FUNCTION "FC_Any_ASCII_To_DInt" : VOID
TITLE =%version: 0.06 % CN: 31
//Function:
//Convert a field of ASCII digits to a Double Integer.
//
//Description:
//
//IMPORTANT
//When u use symbolics at the input of type ANY that refer to a variable of the
//type array or structure be aware that the number of array or structure is even
//!
//
//examples: array[1..2]; array[1..4]; array[1..24]; etc.
//
//             t_char   STRUCT
//              |nr_1   BYTE
//              |nr_2   BYTE
//              |nr_3   BYTE
//              |nr_4   BYTE
//
//The any pointer i_ASCII_pnt points to an area which contains an ASCII number.
//When called, this function converts the imported ASCII-number to a double
//integer and returns the result through o_DInteger_number. The ASCII number can
//be of 1 up to 10 bytes. The ASCII number is split into three double integer
//parts. Then the three parts are checked on the physical limit of a double
//integer. This results into an input specification a range of 0..2147483647.
//When the ASCII-number is out of range, the conversion will not be carried out*.
//Contents of the address registers are being remembered during the block call.
//This way the address registers can be used in the current block.
//The output o_RET_VAL contains information about the cause of the errror.
//· Code 0000:
//No error.
//· Code 3115: {information code}
//The area destination of the any pointer is too small (<5 bytes). When the
//integer number is greater than the destination, only the msb's of the integer
//number will be copied.
//. Code 3112: {error code}
//ASCII type is not 3x hex (0 <= x <=  9). BR-bit is set.
//. Code 3111: {error code}
//The double integer number is out of range. BR-bit is set.
//. Code 3113: {error code}
//Data type is neither byte nor char. BR-bit is set.
//. Code 3114: {error code}
//Wrong memory area from any pointer. BR-bit is set.
//
//
//example: '1248365402' (31 32 34 38 33 36 35 34 30 32 hex.)is converted
//into 1248365402
//
//History:
//This version  %created_by:   %
//              %date_created:   %
//              %release: ECS_General_PLC/dev %
//
//Initial version based on the FC_Any_ASCII_To_DInt Rev: 1.11 of the SSS General
//library
//
//Modification History:                                   By:    Date:     Rev:
//----------------------------------------------------  -------  --------  -----
//7324: ECS-P General from the RD to RA for platform    nlHdL    06-07-15   0.06
//15807: Block consistency update IO symbols, comment   nlHdL    18-09-13   0.06
//CR8255 Update internal logging event value            nlcsu    11-11-11   0.05
//CR6415 Remove o_RET_VAL                               nlple    28-09-11   0.04
//CR6341 Update to coding standard                      nlHdL    27-01-11   0.03
//CR6275 Changing compilation number                    nlple    17-01-11   0.02
//Initial revision                                      nlple    14-01-11   0.01
//
FAMILY : General
VERSION : 0.0


VAR_INPUT
  i_ANY_ASCII : ANY ;	//ANY pointer to the ASCII digits
  i_DB_Event_Num : INT ;	//Number of DB event
END_VAR
VAR_OUTPUT
  o_DINT : DINT ;	//Output of the DINT
END_VAR
VAR_TEMP
  t_char : STRUCT 	//Local Copy of the ASCII digits
   nr_1 : BYTE ;
   nr_2 : BYTE ;
   nr_3 : BYTE ;
   nr_4 : BYTE ;
   nr_5 : BYTE ;
   nr_6 : BYTE ;
   nr_7 : BYTE ;
   nr_8 : BYTE ;
   nr_9 : BYTE ;
   nr_10 : BYTE ;
  END_STRUCT ;
  t_DInteger_H : DINT ;	//Double Integer High part: Bytes 1..4
  t_DInteger_M : DINT ;	//Double Integer Medium part: Bytes 5..8
  t_DInteger_L : DINT ;	//Double Integer Low part: Bytes 9..10
  t_ANY_P_ASCII : ANY ;	//Temp of the ANY pointer
  t_DInteger_number : DINT ;	//Temp of Double Integer
  t_ANY_P_Byte_Address : INT ;	//Byte Address of ANY
  t_Data_Type : DWORD ;	//Data Type of ANY
  t_ANY_P_Length : INT ;	//Lenght of ANY
  t_AR1_Store : DWORD ;	//Store for AR1
  t_AR2_Store : DWORD ;	//Store for AR2
  t_Loop_cntr : INT ;	//Loop Counter
  t_Data_Type_Byte : BYTE ;	//Date Type
  t_DB_Number : INT ;	//DataBlock Number
  t_integer : INT ;	//Integer for storage of data
  t_AR1_Memory : DWORD ;
  t_AR2_Memory : DWORD ;
  t_Ret_Event : INT ;	//Return value for Write Event
END_VAR
BEGIN
NETWORK
TITLE =AA: store address registers and preset return value
//The address registers are used in this block. In this network the address
//registers are stored to be remembered. The return value of this function is
//presetted on zero.
      TAR1  ; //Store AR1
      T     #t_AR1_Store;
      TAR2  ; //Store AR2
      T     #t_AR2_Store;
NETWORK
TITLE =BA: check any pointer
//The any pointer is checked on data type and memory area. And further
//information is stored to be used later in the program.
      L     P##i_ANY_ASCII; //input any pointer
      LAR1  ;

//check data type on byte
      O(    ;
      L     B [AR1,P#1.0];
      L     B#16#2;
      ==I   ; //IF data type =byte
      )     ;
      O(    ;
      L     B [AR1,P#1.0];
      L     B#16#3;
      ==I   ; //IF data type =char
      )     ;
      JC    BA01; //THEN copy any pointer
      SET   ; //set RLO-bit
      SAVE  ; //save RLO status in BR-bit

      L     B [AR1,P#1.0];
      T     #t_integer;

      CALL "FC_Write_Event" (// Report event "Data type ANY pointer is incorrect" (3116)
           i_Message_ID             := 3116,
           i_Event_value            := #t_integer,
           i_DB_Event_Num           := #i_DB_Event_Num,
           o_Return_Value           := #t_Ret_Event);

      JU    HA01;

BA01: L     W [AR1,P#2.0]; //load byte 2&3 = message length
      T     #t_ANY_P_Length; //store message length
      L     W [AR1,P#4.0]; //load byte 4&5 = DB number
      T     #t_DB_Number; //store DB number
      A(    ;
      L     W#16#0;
      >I    ; //IF1 DB pointer
      )     ;
      JCN   BA03; //ELSE1 do not open DB or DI
      A(    ; //THEN1:
      L     B [AR1,P#6.0];
      L     B#16#84;
      ==I   ; //IF2 memory area = DB
      )     ;
      JCN   BA02;
      OPN   DB [#t_DB_Number]; //THEN2 open DB
      JU    BA03;

BA02: OPN   DI [#t_DB_Number]; //ELSE2 open DI

BA03: L     B [AR1,P#6.0]; //load area code of crossing pointer
      T     #t_Data_Type_Byte; //store data type (byte)
      SLD   24;
      T     #t_Data_Type; //store data type for area pointer
      L     D [AR1,P#6.0]; //load area crossing pointer
      AD    DW#16#FFFF; //mask address area
      SRD   3; //remove bit address from accu 1
      T     #t_ANY_P_Byte_Address; //store begin byte address
NETWORK
TITLE =CA: create destination and source pointer
//Depending on the length of the destination area destination and source pointers
//are being created. IF length>=10 THEN source pointer reserves a 10 byte space
//in the destination area ELSE only msb's of the integer are copied
//
      L     #t_ANY_P_Length;
      L     10;
      >=I   ; //IF1 length >= 10
      JCN   CA01;

//create source pointer
      L     #t_ANY_P_Length;
      L     10;
      T     #t_Loop_cntr; //set loop counter
      -I    ;
      L     #t_ANY_P_Byte_Address;
      +I    ;
      ITD   ;
      SLD   3;
      L     #t_Data_Type;
      +D    ;
      LAR2  ;

//create destination pointer
      L     P##t_char;
      LAR1  ; // store source pointer in AR1
      JU    CA99;

//ELSE1 length < 10
CA01: L     DW#16#30303030;
      T     LD     0; //reset t_char.nr_1..4
      L     DW#16#30303030;
      T     LD     4; //reset t_char.nr_5..8
      L     W#16#3030;
      T     LW     8; //reset t_char.nr_9..10

//create source pointer
      L     D [AR1,P#6.0];
      LAR2  ;

//create destination pointer
      L     10;
      L     #t_ANY_P_Length;
      T     #t_Loop_cntr;
      -I    ;
      SLW   3;
      L     DW#16#86000000;
      OD    ;
      LAR1  ;

      TAR1  #t_AR1_Memory; //Store Address Registers
      TAR2  #t_AR2_Memory;

      CALL "FC_Write_Event" (// Report event "Area destination of the ANY pointer is too small" (3115)
           i_Message_ID             := 3115,
           i_Event_value            := #t_ANY_P_Length,
           i_DB_Event_Num           := #i_DB_Event_Num,
           o_Return_Value           := #t_Ret_Event);

      LAR1  #t_AR1_Memory; //Restore Address Registers
      LAR2  #t_AR2_Memory;

CA99: NOP   0;
NETWORK
TITLE =DA: copy contents of i_ANY_P_ASCII
//Copy bytes from source area to local data area.
//CASE t_Data_Type_Byte OF
      L     #t_Data_Type_Byte;
      L     B#16#83;
      ==I   ; //1: t_Data_Type_Byte = 83
      L     #t_Loop_cntr;
      JC    DA01; //copy from memory bits memory area
      L     #t_Data_Type_Byte;
      L     B#16#84;
      ==I   ; //2: t_Data_Type_Byte = 84
      L     #t_Loop_cntr;
      JC    DA02; //copy from data block
      L     #t_Data_Type_Byte;
      L     B#16#85;
      ==I   ; //3: t_Data_Type_Byte = 85
      L     #t_Loop_cntr;
      JC    DA03; //copy from instance data block
      L     #t_Data_Type_Byte;
      L     B#16#87;
      ==I   ; //4: t_Data_Type_Byte = 87
      L     #t_Loop_cntr;
      JC    DA04; //copy from previous local data
      SET   ; //set RLO-bit
      SAVE  ; //save RLO status in BR-bit

      L     #t_Data_Type_Byte;
      T     #t_integer;

      CALL "FC_Write_Event" (// Report event "The ANY pointer has a wrong memory area" (3114)
           i_Message_ID             := 3114,
           i_Event_value            := #t_integer,
           i_DB_Event_Num           := #i_DB_Event_Num,
           o_Return_Value           := #t_Ret_Event);

      JU    HA01;

DA01: T     #t_Loop_cntr;
      L     MB [AR2,P#0.0];
      T     LB [AR1,P#0.0];
      +AR1  P#1.0;
      +AR2  P#1.0;
      L     #t_Loop_cntr;
      LOOP  DA01;
      JU    DA05;

DA02: T     #t_Loop_cntr;
      L     DBB [AR2,P#0.0];
      T     LB [AR1,P#0.0];
      +AR1  P#1.0;
      +AR2  P#1.0;
      L     #t_Loop_cntr;
      LOOP  DA02;
      JU    DA05;

DA03: T     #t_Loop_cntr;
      L     DIB [AR2,P#0.0];
      T     LB [AR1,P#0.0];
      +AR1  P#1.0;
      +AR2  P#1.0;
      L     #t_Loop_cntr;
      LOOP  DA03;
      JU    DA05;

DA04: T     #t_Loop_cntr;
      L     B [AR2,P#0.0];
      T     LB [AR1,P#0.0];
      +AR1  P#1.0;
      +AR2  P#1.0;
      L     #t_Loop_cntr;
      LOOP  DA04;

DA05: NOP   0;
NETWORK
TITLE =EA: check ASCII type & split ASCII into parts
//Check if the ASCII type = 3hex.
//Convert ASCII-number into three double integer parts: t_DInteger High, Middle
//and Low part.
//check ASCII type
      L     LD     0; //load ASCII char 1..4
      L     DW#16#F0F0F0F0;
      AD    ;
      A(    ;
      L     DW#16#30303030;
      ==D   ; //IF ASCII type = 30 hex
      )     ;

      L     LD     4; //load ASCII char 5..8
      L     DW#16#F0F0F0F0;
      AD    ;
      A(    ;
      L     DW#16#30303030;
      ==D   ; //ANDIF ASCII type = 30 hex
      )     ;

      L     LW     8; //load ASCII char 9..10
      L     DW#16#F0F0;
      AW    ;
      A(    ;
      L     DW#16#3030;
      ==D   ; //ANDIF ASCII type = 30 hex
      )     ;
      JC    EA01; //THEN filter hex30
      SET   ; //set RLO-bit
      SAVE  ; //save RLO status in BR-bit

      CALL "FC_Write_Event" (// Report event 'Data_Type_Conversion: ASCII character(s) out of range (0 <= X <= 9)' (3112)
           i_Message_ID             := 3112,
           i_Event_value            := 1,
           i_DB_Event_Num           := #i_DB_Event_Num,
           o_Return_Value           := #t_Ret_Event);

      JU    HA01;

//filter ASCII number
EA01: L     LD     0; //load ASCII-number for conversion
      L     DW#16#F0F0F0F;
      AD    ; //filter hex30
      T     LD     0;

      L     LD     4; //load ASCII-number for conversion
      L     DW#16#F0F0F0F;
      AD    ; //filter hex30
      T     LD     4;

      L     LW     8; //load ASCII-number for conversion
      L     W#16#F0F;
      AW    ; //filter hex30
      T     LW     8;

//split ASCII number into 3 DIntegers
      L     #t_char.nr_1; //load milliards
      L     10;
      *D    ; //multiply with 10
      L     #t_char.nr_2; //load hundred millions
      +D    ; //add accu1 + hundred millions
      L     10;
      *D    ; //multiply with 10
      L     #t_char.nr_3; //load ten millions
      +D    ; //add accu1 + ten millions
      L     10;
      *D    ; //multiply with 10
      L     #t_char.nr_4; //load millions
      +D    ; //add accul + millions
      T     #t_DInteger_H; //high number part

      L     #t_char.nr_5; //load hundred thousands
      L     10;
      *D    ; //multiply with 10
      L     #t_char.nr_6; //load ten thousands
      +D    ; //add accu1 + ten thousands
      L     10;
      *D    ; //multiply with 10
      L     #t_char.nr_7; //load thousands
      +D    ; //add accu1 + thousands
      L     10;
      *D    ; //multiply with 10
      L     #t_char.nr_8; //load hundreds
      +D    ; //add accu1 + hundreds
      T     #t_DInteger_M; //middle number part

      L     #t_char.nr_9; //load tens
      L     10;
      *D    ; //multiply with 10
      L     #t_char.nr_10; //load units
      +D    ; //add accu1 + units
      T     #t_DInteger_L; //low number part
NETWORK
TITLE =FA: check ASCII number
//Checks input ASCII number on range.
//ASCII must be between 0 and +2147483647. If not, RLO = 0 and there is no
//conversion.
      A(    ;
      L     #t_DInteger_H;
      L     2147;
      ==D   ; //IF1 t_DInteger_H =2147
      )     ;
      JCN   FA01;
      A(    ; //THEN1
      L     #t_DInteger_M;
      L     4836;
      ==D   ; //IF2 t_DInteger_M =4836
      )     ;
      JCN   FA02;
      JU    FA03;
FA01: A(    ; //ELSE1
      L     #t_DInteger_H;
      L     2147;
      <D    ; //IF3 t_DInteger_H <2147
      )     ;
      JCN   FA04;
      JU    FA05;
FA02: A(    ; //THEN2
      L     #t_DInteger_M;
      L     4836;
      <D    ; //IF4 t_DInteger_M <4836
      )     ;
      JCN   FA04;
      JU    FA05;
FA03: A(    ; //ELSE2
      L     #t_DInteger_L;
      L     47;
      <=D   ; //IF5  t_DInteger_L <=47
      )     ;
      JCN   FA05;
FA04: SET   ; //set RLO-bit
      SAVE  ; //save RLO status in BR-bit

      CALL "FC_Write_Event" (// Report event 'Data_Type_Conversion: ASCII character(s) out of range (0 <= X <= 9)' (3112)
           i_Message_ID             := 3112,
           i_Event_value            := 1,
           i_DB_Event_Num           := #i_DB_Event_Num,
           o_Return_Value           := #t_Ret_Event);


      JU    HA01;
FA05: NOP   0;
NETWORK
TITLE =GA: convert ASCII to DINT
//After a correct ceck, the already coverted parts will be converted into a
//double
//integer.
      L     #t_DInteger_H;
      L     L#1000000;
      *D    ;
      T     #t_DInteger_number;

      L     #t_DInteger_M;
      L     100;
      *D    ;
      L     #t_DInteger_number;
      +D    ;
      L     #t_DInteger_L;
      +D    ;
      T     #t_DInteger_number;

      L     #t_DInteger_number;
      T     #o_DINT;
NETWORK
TITLE =HA: restore stored address registers
//The stored adderss registers are restored in this network.
HA01: L     #t_AR1_Store;
      LAR1  ;
      L     #t_AR2_Store;
      LAR2  ;
END_FUNCTION

